TYPE ST_Contactor_HMI :
    STRUCT
        Config  : ST_Contactor_Config;
        Command : ST_Contactor_Command;
        Status  : ST_Contactor_Status;
    END_STRUCT
END_TYPE

(* stored: Version 1.1.0.1, ProductVersion 3.1.4024.15
   DUT ST_Contactor_HMI: Id {68e606df-c44a-4278-8523-c23f349863d2} *)
